// Mitsubishi GX Works2 project: 완성본   PLC: Q03UDE

PROGRAM MAIN
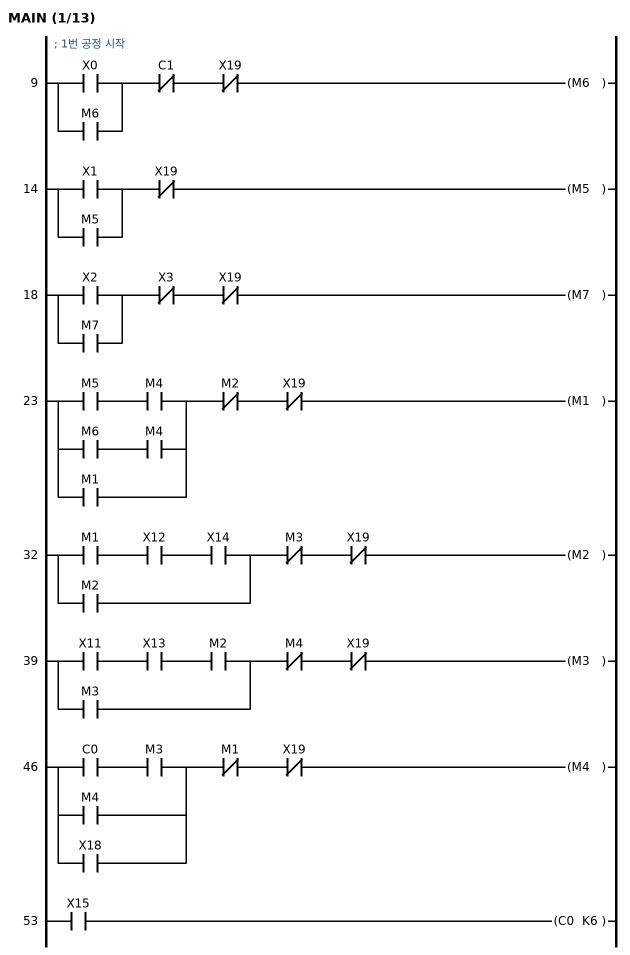
; 1번 공정 시작
9     LD      X0
      OR      M6
      ANI     C1
      ANI     X19
      OUT     M6
14    LD      X1
      OR      M5
      ANI     X19
      OUT     M5
18    LD      X2
      OR      M7
      ANI     X3
      ANI     X19
      OUT     M7
23    LD      M5
      AND     M4
      LD      M6
      AND     M4
      ORB
      OR      M1
      ANI     M2
      ANI     X19
      OUT     M1
32    LD      M1
      AND     X12
      AND     X14
      OR      M2
      ANI     M3
      ANI     X19
      OUT     M2
39    LD      X11
      AND     X13
      AND     M2
      OR      M3
      ANI     M4
      ANI     X19
      OUT     M3
46    LD      C0
      AND     M3
      OR      M4
      OR      X18
      ANI     M1
      ANI     X19
      OUT     M4
53    LD      X15
      OUT     C0 K6
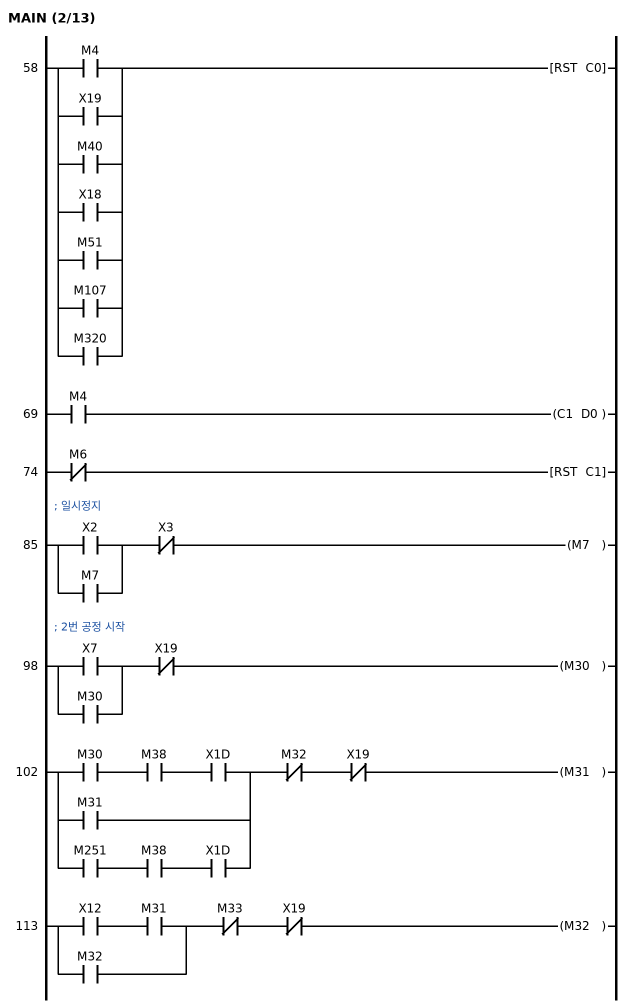
58    LD      M4
      OR      X19
      OR      M40
      OR      X18
      OR      M51
      OR      M107
      OR      M320
      RST     C0
69    LD      M4
      OUT     C1 D0
74    LDI     M6
      RST     C1
; 일시정지
85    LD      X2
      OR      M7
      ANI     X3
      OUT     M7
; 2번 공정 시작
98    LD      X7
      OR      M30
      ANI     X19
      OUT     M30
102   LD      M30
      AND     M38
      AND     X1D
      OR      M31
      LD      M251
      AND     M38
      AND     X1D
      ORB
      ANI     M32
      ANI     X19
      OUT     M31
113   LD      X12
      AND     M31
      OR      M32
      ANI     M33
      ANI     X19
      OUT     M32
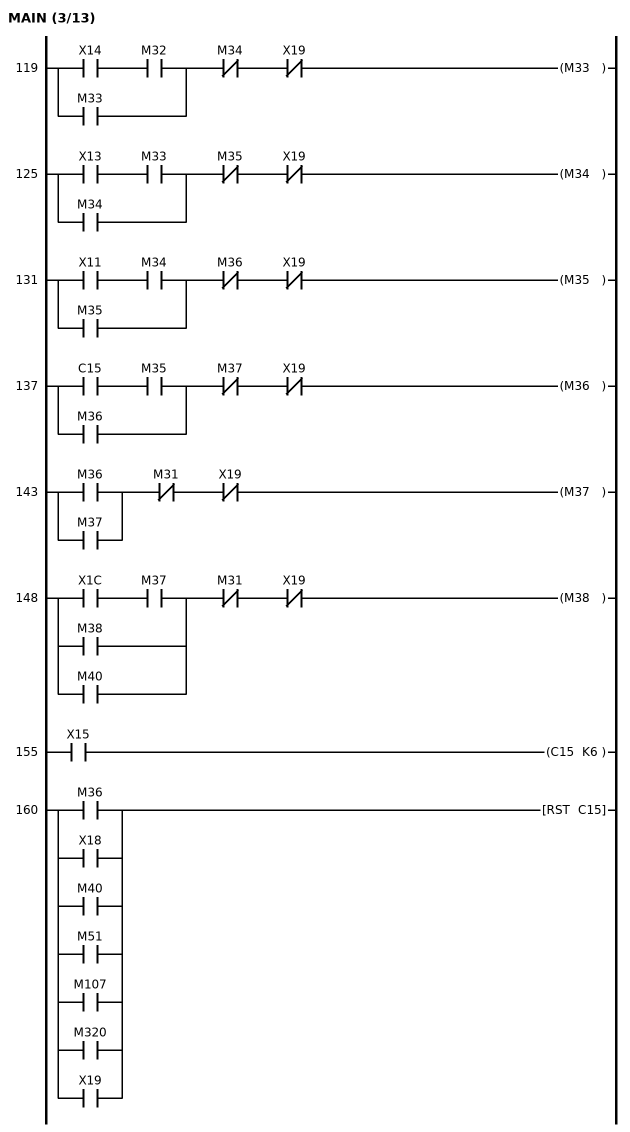
119   LD      X14
      AND     M32
      OR      M33
      ANI     M34
      ANI     X19
      OUT     M33
125   LD      X13
      AND     M33
      OR      M34
      ANI     M35
      ANI     X19
      OUT     M34
131   LD      X11
      AND     M34
      OR      M35
      ANI     M36
      ANI     X19
      OUT     M35
137   LD      C15
      AND     M35
      OR      M36
      ANI     M37
      ANI     X19
      OUT     M36
143   LD      M36
      OR      M37
      ANI     M31
      ANI     X19
      OUT     M37
148   LD      X1C
      AND     M37
      OR      M38
      OR      M40
      ANI     M31
      ANI     X19
      OUT     M38
155   LD      X15
      OUT     C15 K6
160   LD      M36
      OR      X18
      OR      M40
      OR      M51
      OR      M107
      OR      M320
      OR      X19
      RST     C15
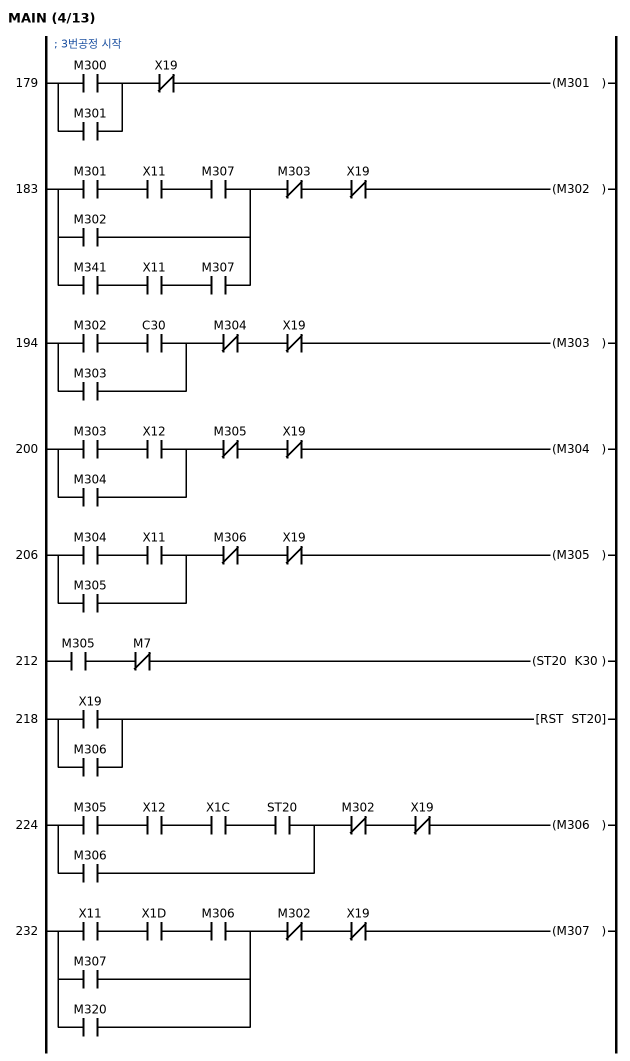
; 3번공정 시작
179   LD      M300
      OR      M301
      ANI     X19
      OUT     M301
183   LD      M301
      AND     X11
      AND     M307
      OR      M302
      LD      M341
      AND     X11
      AND     M307
      ORB
      ANI     M303
      ANI     X19
      OUT     M302
194   LD      M302
      AND     C30
      OR      M303
      ANI     M304
      ANI     X19
      OUT     M303
200   LD      M303
      AND     X12
      OR      M304
      ANI     M305
      ANI     X19
      OUT     M304
206   LD      M304
      AND     X11
      OR      M305
      ANI     M306
      ANI     X19
      OUT     M305
212   LD      M305
      ANI     M7
      OUT     ST20 K30
218   LD      X19
      OR      M306
      RST     ST20
224   LD      M305
      AND     X12
      AND     X1C
      AND     ST20
      OR      M306
      ANI     M302
      ANI     X19
      OUT     M306
232   LD      X11
      AND     X1D
      AND     M306
      OR      M307
      OR      M320
      ANI     M302
      ANI     X19
      OUT     M307
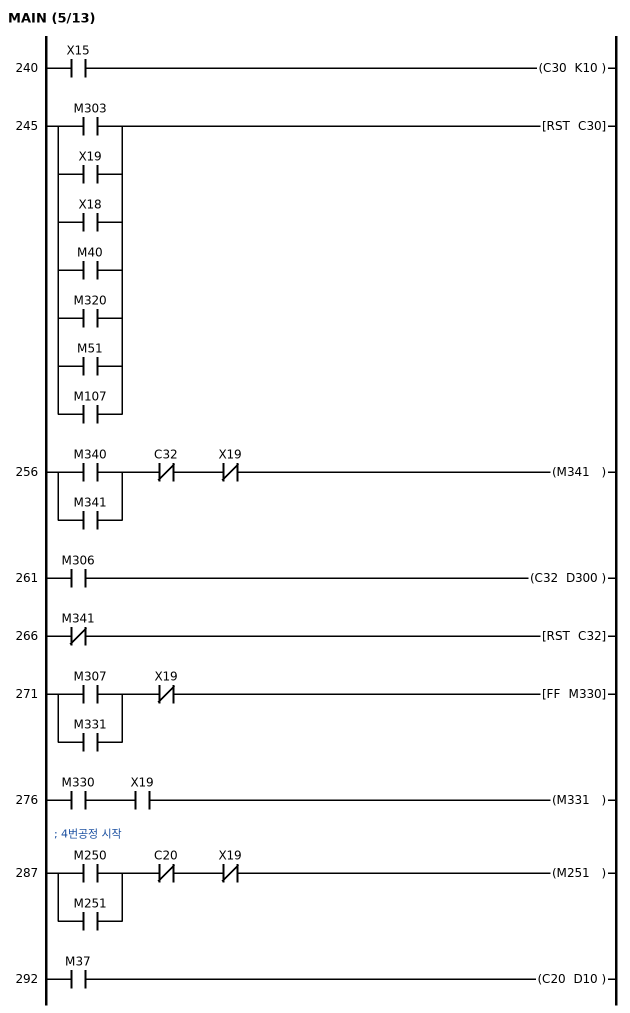
240   LD      X15
      OUT     C30 K10
245   LD      M303
      OR      X19
      OR      X18
      OR      M40
      OR      M320
      OR      M51
      OR      M107
      RST     C30
256   LD      M340
      OR      M341
      ANI     C32
      ANI     X19
      OUT     M341
261   LD      M306
      OUT     C32 D300
266   LDI     M341
      RST     C32
271   LD      M307
      OR      M331
      ANI     X19
      FF      M330
276   LD      M330
      AND     X19
      OUT     M331
; 4번공정 시작
287   LD      M250
      OR      M251
      ANI     C20
      ANI     X19
      OUT     M251
292   LD      M37
      OUT     C20 D10
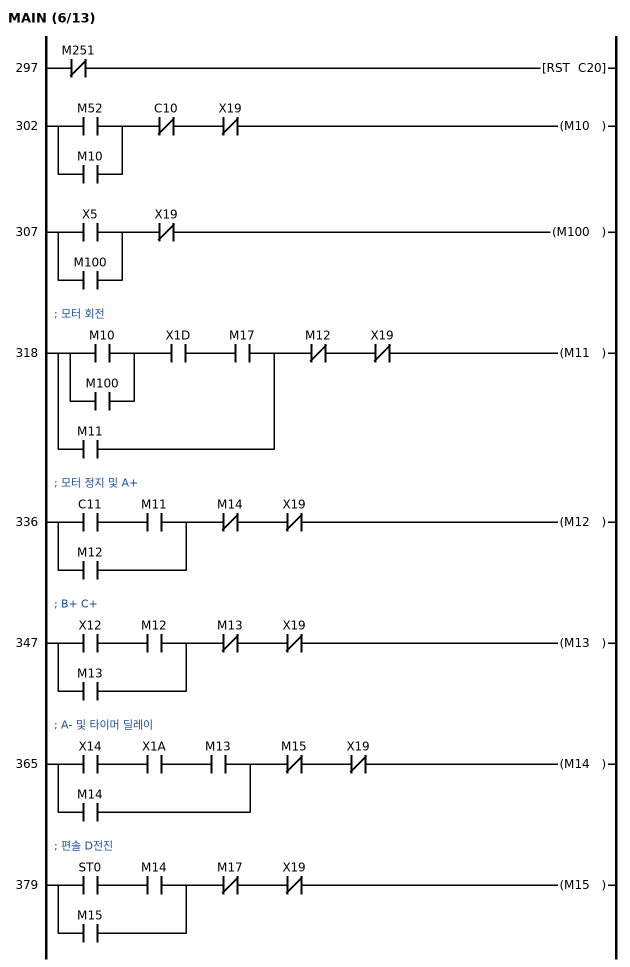
297   LDI     M251
      RST     C20
302   LD      M52
      OR      M10
      ANI     C10
      ANI     X19
      OUT     M10
307   LD      X5
      OR      M100
      ANI     X19
      OUT     M100
; 모터 회전
318   LD      M10
      OR      M100
      AND     X1D
      AND     M17
      OR      M11
      ANI     M12
      ANI     X19
      OUT     M11
; 모터 정지 및 A+
336   LD      C11
      AND     M11
      OR      M12
      ANI     M14
      ANI     X19
      OUT     M12
; B+ C+
347   LD      X12
      AND     M12
      OR      M13
      ANI     M13
      ANI     X19
      OUT     M13
; A- 및 타이머 딜레이
365   LD      X14
      AND     X1A
      AND     M13
      OR      M14
      ANI     M15
      ANI     X19
      OUT     M14
; 편솔 D전진
379   LD      ST0
      AND     M14
      OR      M15
      ANI     M17
      ANI     X19
      OUT     M15
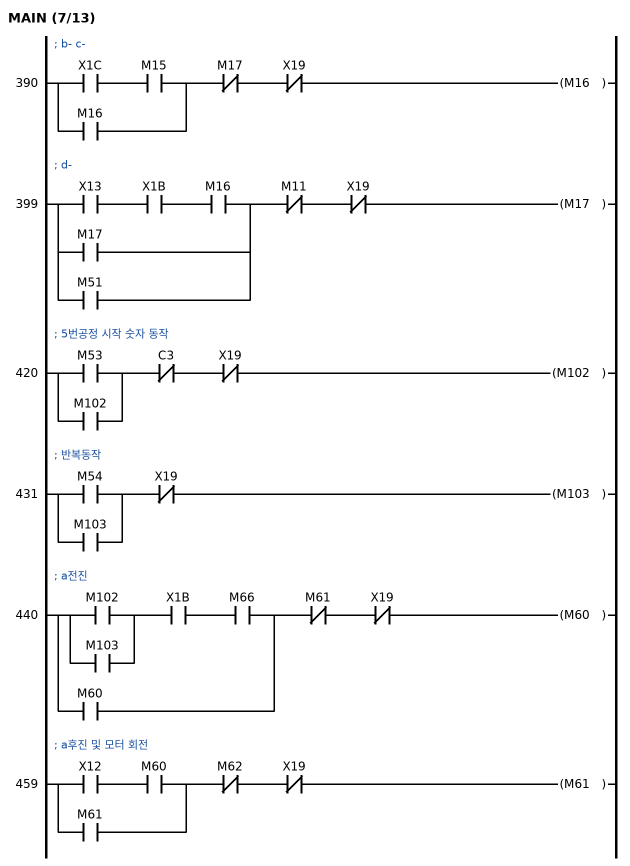
; b- c-
390   LD      X1C
      AND     M15
      OR      M16
      ANI     M17
      ANI     X19
      OUT     M16
; d-
399   LD      X13
      AND     X1B
      AND     M16
      OR      M17
      OR      M51
      ANI     M11
      ANI     X19
      OUT     M17
; 5번공정 시작 숫자 동작
420   LD      M53
      OR      M102
      ANI     C3
      ANI     X19
      OUT     M102
; 반복동작
431   LD      M54
      OR      M103
      ANI     X19
      OUT     M103
; a전진
440   LD      M102
      OR      M103
      AND     X1B
      AND     M66
      OR      M60
      ANI     M61
      ANI     X19
      OUT     M60
; a후진 및 모터 회전
459   LD      X12
      AND     M60
      OR      M61
      ANI     M62
      ANI     X19
      OUT     M61
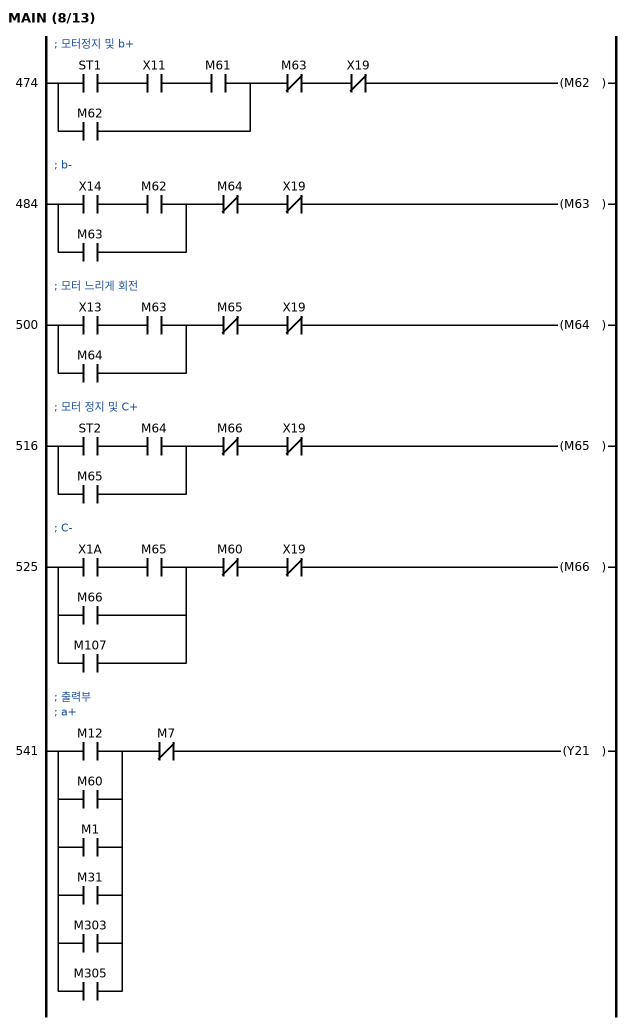
; 모터정지 및 b+
474   LD      ST1
      AND     X11
      AND     M61
      OR      M62
      ANI     M63
      ANI     X19
      OUT     M62
; b-
484   LD      X14
      AND     M62
      OR      M63
      ANI     M64
      ANI     X19
      OUT     M63
; 모터 느리게 회전
500   LD      X13
      AND     M63
      OR      M64
      ANI     M65
      ANI     X19
      OUT     M64
; 모터 정지 및 C+
516   LD      ST2
      AND     M64
      OR      M65
      ANI     M66
      ANI     X19
      OUT     M65
; C-
525   LD      X1A
      AND     M65
      OR      M66
      OR      M107
      ANI     M60
      ANI     X19
      OUT     M66
; 출력부
; a+
541   LD      M12
      OR      M60
      OR      M1
      OR      M31
      OR      M303
      OR      M305
      ANI     M7
      OUT     Y21
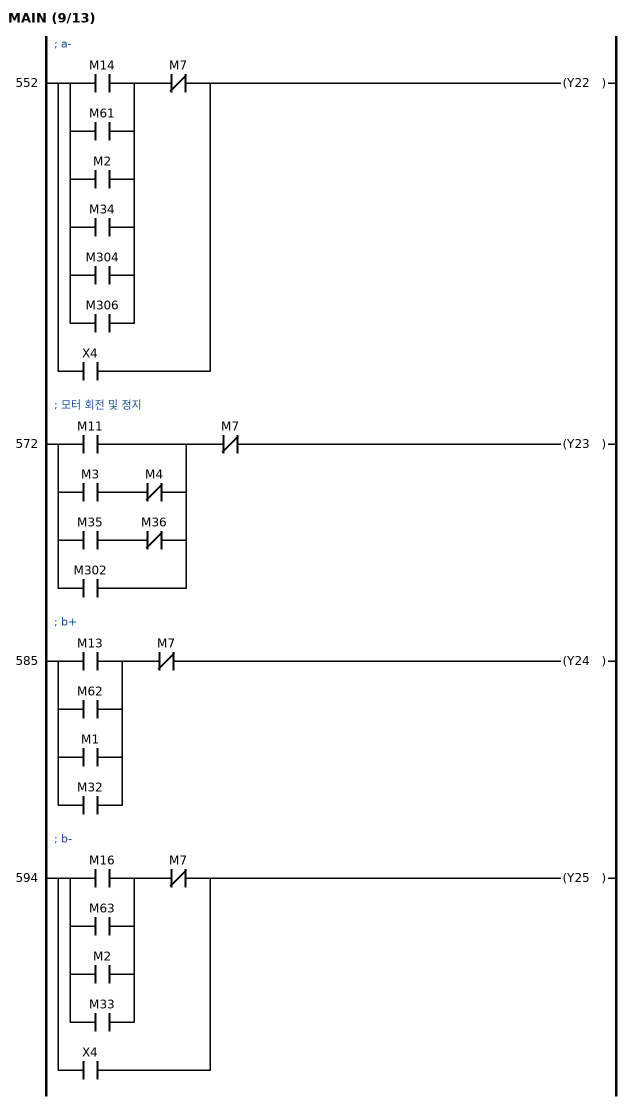
; a-
552   LD      M14
      OR      M61
      OR      M2
      OR      M34
      OR      M304
      OR      M306
      ANI     M7
      OR      X4
      OUT     Y22
; 모터 회전 및 정지
572   LD      M11
      LD      M3
      ANI     M4
      ORB
      LD      M35
      ANI     M36
      ORB
      OR      M302
      ANI     M7
      OUT     Y23
; b+
585   LD      M13
      OR      M62
      OR      M1
      OR      M32
      ANI     M7
      OUT     Y24
; b-
594   LD      M16
      OR      M63
      OR      M2
      OR      M33
      ANI     M7
      OR      X4
      OUT     Y25
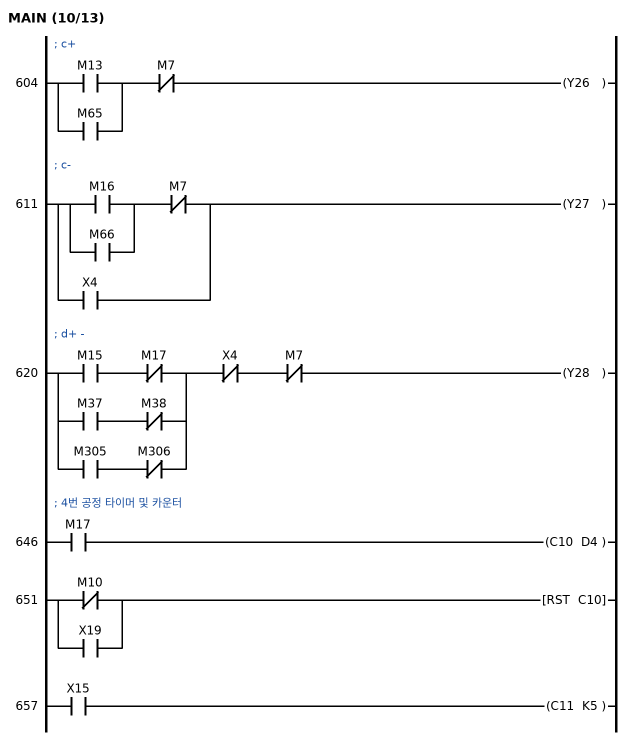
; c+
604   LD      M13
      OR      M65
      ANI     M7
      OUT     Y26
; c-
611   LD      M16
      OR      M66
      ANI     M7
      OR      X4
      OUT     Y27
; d+ -
620   LD      M15
      ANI     M17
      LD      M37
      ANI     M38
      ORB
      LD      M305
      ANI     M306
      ORB
      ANI     X4
      ANI     M7
      OUT     Y28
; 4번 공정 타이머 및 카운터
646   LD      M17
      OUT     C10 D4
651   LDI     M10
      OR      X19
      RST     C10
657   LD      X15
      OUT     C11 K5
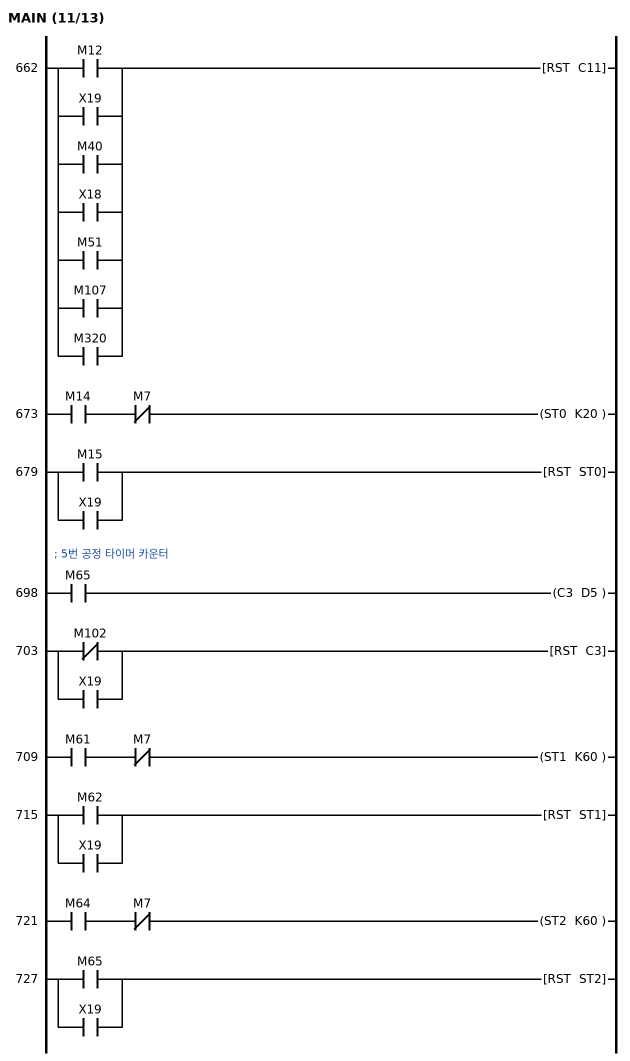
662   LD      M12
      OR      X19
      OR      M40
      OR      X18
      OR      M51
      OR      M107
      OR      M320
      RST     C11
673   LD      M14
      ANI     M7
      OUT     ST0 K20
679   LD      M15
      OR      X19
      RST     ST0
; 5번 공정 타이머 카운터
698   LD      M65
      OUT     C3 D5
703   LDI     M102
      OR      X19
      RST     C3
709   LD      M61
      ANI     M7
      OUT     ST1 K60
715   LD      M62
      OR      X19
      RST     ST1
721   LD      M64
      ANI     M7
      OUT     ST2 K60
727   LD      M65
      OR      X19
      RST     ST2
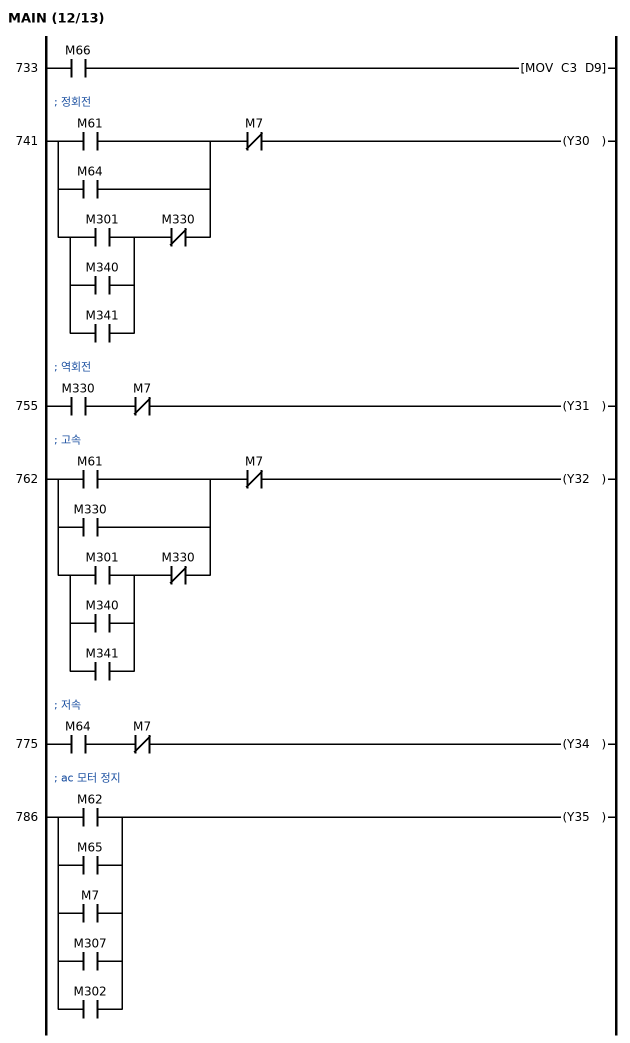
733   LD      M66
      MOV     C3 D9
; 정회전
741   LD      M61
      OR      M64
      LD      M301
      OR      M340
      OR      M341
      ANI     M330
      ORB
      ANI     M7
      OUT     Y30
; 역회전
755   LD      M330
      ANI     M7
      OUT     Y31
; 고속
762   LD      M61
      OR      M330
      LD      M301
      OR      M340
      OR      M341
      ANI     M330
      ORB
      ANI     M7
      OUT     Y32
; 저속
775   LD      M64
      ANI     M7
      OUT     Y34
; ac 모터 정지
786   LD      M62
      OR      M65
      OR      M7
      OR      M307
      OR      M302
      OUT     Y35
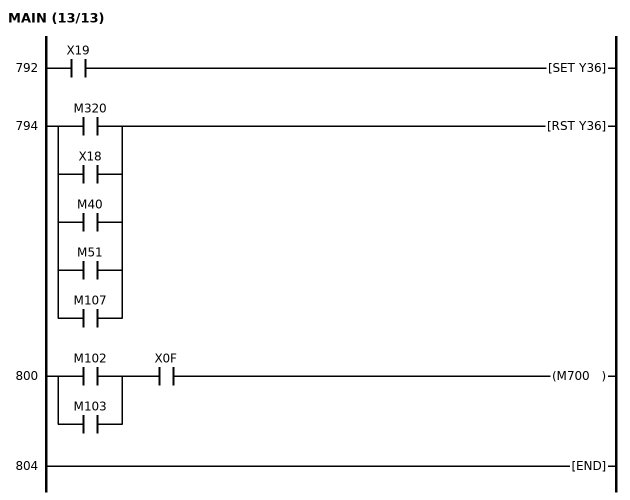
792   LD      X19
      SET     Y36
794   LD      M320
      OR      X18
      OR      M40
      OR      M51
      OR      M107
      RST     Y36
800   LD      M102
      OR      M103
      AND     X0F
      OUT     M700
804   END
END_PROGRAM
